PROGRAM BackgroundEL
VAR
	(* background communication with the EL6001/EL6002 terminal *)
	afbEL6002Ctrl			: ARRAY[gc.MINDEVICEINDEX..gc.MAXDEVICEINDEX] OF SerialLineControl;
	abEL6002CtrlError		: ARRAY[gc.MINDEVICEINDEX..gc.MAXDEVICEINDEX] OF BOOL;
	aeEL6002CtrlErrorID		: ARRAY[gc.MINDEVICEINDEX..gc.MAXDEVICEINDEX] OF ComError_t;
	(* 	I/O variables for a EL6001 terminal*)
	astIn_EL6002 AT %I*		: ARRAY[gc.MINDEVICEINDEX..gc.MAXDEVICEINDEX] OF EL6inData22B;	(* linked to the EL6001 in the TwinCAT System Manager *)
	astOut_EL6002 AT %Q*	: ARRAY[gc.MINDEVICEINDEX..gc.MAXDEVICEINDEX] OF EL6outData22B;(* linked to the EL6001 in the TwinCAT System Manager *)
END_VAR

(*
The SerialLineControl function block is supposed to be called in every PLC cycle.
It communicates with the serial line hardware device and transmits or receives data.
The SerialLineControl can be called in the standard task (e.g.for PcCOM port usage) 
or in a separate fast task (e.g.for terminal usage) as well.
A fast separate task will be necessary at high baud rates or with KL6001 terminals 
which have a small process image (3 or 5 data bytes only)
*)

(* background communication with the EL6002 terminal *)

//use with type SerialLineControl
afbEL6002Ctrl[gc.EL6002_INDEX1](
	Mode:= SERIALLINEMODE_EL6_22B, 
	pComIn:= ADR(astIn_EL6002[gc.EL6002_INDEX1]), 
	pComOut:= ADR(astOut_EL6002[gc.EL6002_INDEX1]), 
	SizeComIn:= SIZEOF(astIn_EL6002[gc.EL6002_INDEX1]), 
	Error=> , 
	ErrorID=> , 
	TxBuffer:= aTxBufferEL[gc.EL6002_INDEX1], 
	RxBuffer:= aRxBufferEL[gc.EL6002_INDEX1] );
IF afbEL6002Ctrl[gc.EL6002_INDEX1].Error THEN
	abEL6002CtrlError[gc.EL6002_INDEX1] := TRUE;
	aeEL6002CtrlErrorID[gc.EL6002_INDEX1] := afbEL6002Ctrl[gc.EL6002_INDEX1].ErrorID;
END_IF

END_PROGRAM

(* stored: Version 1.1.0.1, ProductVersion 3.1.4024.9
   POU BackgroundEL: Id {9a20473f-0d3f-4584-b429-33e10587a848}, SpecialFunc None *)
